(* IEC 61131-3 sources: PLC61131Repos/BZ172Lab/HMIRemote (part 2) *)

	UNTIL pagID <> 16#00
	END_REPEAT;

END_FUNCTION_BLOCK

FUNCTION_BLOCK RefrUnit

	VAR_EXTERNAL
	guiCallStack : ARRAY[ 0..9 ] OF UINT;
	giStackPtr : INT;
	fbUnitString_10 : Static01;
	fbUnitEdit_9 : EditBox01;
	fbUnitEdit_12 : EditBox01;
	fbUnitEdit_13 : EditBox01;
	fbUnitEdit_14 : EditBox01;
	fbUnitEdit_15 : EditBox01;
	fbRefrEvaporatorFan : RefrEvaporatorFan;
	$waitRefresh : BOOL;
	END_VAR

	VAR
	res : USINT;
	pagID : UINT;
	n : USINT;
	iSP : INT;
	pDC : UDINT;
	rx1 : UINT;
	ry1 : UINT;
	rx2 : UINT;
	ry2 : UINT;
	END_VAR

	{CODE:ST}

	REPEAT

		(* Locking the video *)
		res := Video_Lock( res );

		(* Testing if page has changed *)
		pagID := guiCallStack[ giStackPtr ];

		IF pagID = 16#04 THEN

			(* the refresh task is arrived *)
			$waitRefresh := FALSE;

			(* *** REFRESH PAGE CONTROLS *** *)
			IF fbUnitEdit_9.accMode <> kACS_MODIFY THEN
				fbUnitEdit_9();
			END_IF;
			fbUnitEdit_12();
			fbUnitEdit_13();
			fbUnitEdit_14();
			fbUnitEdit_15();

			(* *** REFRESHING BACKGROUND ITEMS *** *)
			(* Cursor across the call stack *)
			iSP := giStackPtr;

			(* *** REFRESHING PARENT BACKGROUND ITEMS *** *)

		END_IF;

		(* Unlocking the video *)
		res := Video_Unlock( res );

		(* Suspending the task *)
		res := Video_Sleep( 50 );

		(* *** MANAGING CHILD WINDOWS AND ALARM MESSAGES *** *)
		IF pagID <> 16#04 THEN
			CASE pagID OF
				16#02:
					fbRefrEvaporatorFan();

			END_CASE;

			(* Re-testing if this page is active *)
			res := Video_Lock( res );
			pagID := guiCallStack[ giStackPtr ];
			res := Video_Unlock( res );
		END_IF;

	UNTIL pagID <> 16#04
	END_REPEAT;

END_FUNCTION_BLOCK

FUNCTION_BLOCK RefrEvaporatorFan

	VAR_EXTERNAL
	guiCallStack : ARRAY[ 0..9 ] OF UINT;
	giStackPtr : INT;
	fbEvaporatorFanString_10 : Static01;
	fbEvaporatorFanString_11 : Static01;
	fbEvaporatorFanString_12 : Static01;
	fbEvaporatorFanString_13 : Static01;
	fbEvaporatorFanEdit_1 : EditBox01;
	fbEvaporatorFanEdit_2 : EditBox01;
	fbEvaporatorFanEdit_3 : EditBox01;
	fbEvaporatorFanEdit_5 : EditBox01;
	fbEvaporatorFanEdit_6 : EditBox01;
	fbEvaporatorFanEdit_7 : EditBox01;
	fbEvaporatorFanEdit_8 : EditBox01;
	fbEvaporatorFanEdit_9 : EditBox01;
	fbRefrCompressor : RefrCompressor;
	$waitRefresh : BOOL;
	END_VAR

	VAR
	res : USINT;
	pagID : UINT;
	n : USINT;
	iSP : INT;
	pDC : UDINT;
	rx1 : UINT;
	ry1 : UINT;
	rx2 : UINT;
	ry2 : UINT;
	END_VAR

	{CODE:ST}

	REPEAT

		(* Locking the video *)
		res := Video_Lock( res );

		(* Testing if page has changed *)
		pagID := guiCallStack[ giStackPtr ];

		IF pagID = 16#02 THEN

			(* the refresh task is arrived *)
			$waitRefresh := FALSE;

			(* *** REFRESH PAGE CONTROLS *** *)
			IF fbEvaporatorFanEdit_1.accMode <> kACS_MODIFY THEN
				fbEvaporatorFanEdit_1();
			END_IF;
			IF fbEvaporatorFanEdit_2.accMode <> kACS_MODIFY THEN
				fbEvaporatorFanEdit_2();
			END_IF;
			IF fbEvaporatorFanEdit_3.accMode <> kACS_MODIFY THEN
				fbEvaporatorFanEdit_3();
			END_IF;
			IF fbEvaporatorFanEdit_5.accMode <> kACS_MODIFY THEN
				fbEvaporatorFanEdit_5();
			END_IF;
			fbEvaporatorFanEdit_6();
			fbEvaporatorFanEdit_7();
			fbEvaporatorFanEdit_8();
			fbEvaporatorFanEdit_9();

			(* *** REFRESHING BACKGROUND ITEMS *** *)
			(* Cursor across the call stack *)
			iSP := giStackPtr;

			(* *** REFRESHING PARENT BACKGROUND ITEMS *** *)

		END_IF;

		(* Unlocking the video *)
		res := Video_Unlock( res );

		(* Suspending the task *)
		res := Video_Sleep( 50 );

		(* *** MANAGING CHILD WINDOWS AND ALARM MESSAGES *** *)
		IF pagID <> 16#02 THEN
			CASE pagID OF
				16#01:
					fbRefrCompressor();

			END_CASE;

			(* Re-testing if this page is active *)
			res := Video_Lock( res );
			pagID := guiCallStack[ giStackPtr ];
			res := Video_Unlock( res );
		END_IF;

	UNTIL pagID <> 16#02
	END_REPEAT;

END_FUNCTION_BLOCK

FUNCTION_BLOCK RefrCompressor

	VAR_EXTERNAL
	guiCallStack : ARRAY[ 0..9 ] OF UINT;
	giStackPtr : INT;
	fbCompressorString_8 : Static01;
	fbCompressorString_9 : Static01;
	fbCompressorString_10 : Static01;
	fbCompressorString_11 : Static01;
	fbCompressorString_12 : Static01;
	fbCompressorEdit_1 : EditBox01;
	fbCompressorEdit_2 : EditBox01;
	fbCompressorEdit_3 : EditBox01;
	fbCompressorEdit_4 : EditBox01;
	fbCompressorEdit_5 : EditBox01;
	fbCompressorEdit_6 : EditBox01;
	fbCompressorEdit_7 : EditBox01;
	fbRefrEXV : RefrEXV;
	$waitRefresh : BOOL;
	END_VAR

	VAR
	res : USINT;
	pagID : UINT;
	n : USINT;
	iSP : INT;
	pDC : UDINT;
	rx1 : UINT;
	ry1 : UINT;
	rx2 : UINT;
	ry2 : UINT;
	END_VAR

	{CODE:ST}

	REPEAT

		(* Locking the video *)
		res := Video_Lock( res );

		(* Testing if page has changed *)
		pagID := guiCallStack[ giStackPtr ];

		IF pagID = 16#01 THEN

			(* the refresh task is arrived *)
			$waitRefresh := FALSE;

			(* *** REFRESH PAGE CONTROLS *** *)
			IF fbCompressorEdit_1.accMode <> kACS_MODIFY THEN
				fbCompressorEdit_1();
			END_IF;
			IF fbCompressorEdit_2.accMode <> kACS_MODIFY THEN
				fbCompressorEdit_2();
			END_IF;
			fbCompressorEdit_3();
			fbCompressorEdit_4();
			fbCompressorEdit_5();
			fbCompressorEdit_6();
			fbCompressorEdit_7();

			(* *** REFRESHING BACKGROUND ITEMS *** *)
			(* Cursor across the call stack *)
			iSP := giStackPtr;

			(* *** REFRESHING PARENT BACKGROUND ITEMS *** *)

		END_IF;

		(* Unlocking the video *)
		res := Video_Unlock( res );

		(* Suspending the task *)
		res := Video_Sleep( 50 );

		(* *** MANAGING CHILD WINDOWS AND ALARM MESSAGES *** *)
		IF pagID <> 16#01 THEN
			CASE pagID OF
				16#06:
					fbRefrEXV();

			END_CASE;

			(* Re-testing if this page is active *)
			res := Video_Lock( res );
			pagID := guiCallStack[ giStackPtr ];
			res := Video_Unlock( res );
		END_IF;

	UNTIL pagID <> 16#01
	END_REPEAT;

END_FUNCTION_BLOCK

FUNCTION_BLOCK RefrEXV

	VAR_EXTERNAL
	guiCallStack : ARRAY[ 0..9 ] OF UINT;
	giStackPtr : INT;
	fbEXVString_10 : Static01;
	fbEXVString_11 : Static01;
	fbEXVString_12 : Static01;
	fbEXVString_13 : Static01;
	fbEXVString_14 : Static01;
	fbEXVEdit_1 : EditBox01;
	fbEXVEdit_2 : EditBox01;
	fbEXVEdit_4 : EditBox01;
	fbEXVEdit_5 : EditBox01;
	fbEXVEdit_6 : EditBox01;
	fbEXVEdit_7 : EditBox01;
	fbEXVEdit_8 : EditBox01;
	fbEXVEdit_9 : EditBox01;
	fbRefrPIDCoefficients : RefrPIDCoefficients;
	$waitRefresh : BOOL;
	END_VAR

	VAR
	res : USINT;
	pagID : UINT;
	n : USINT;
	iSP : INT;
	pDC : UDINT;
	rx1 : UINT;
	ry1 : UINT;
	rx2 : UINT;
	ry2 : UINT;
	END_VAR

	{CODE:ST}

	REPEAT

		(* Locking the video *)
		res := Video_Lock( res );

		(* Testing if page has changed *)
		pagID := guiCallStack[ giStackPtr ];

		IF pagID = 16#06 THEN

			(* the refresh task is arrived *)
			$waitRefresh := FALSE;

			(* *** REFRESH PAGE CONTROLS *** *)
			IF fbEXVEdit_1.accMode <> kACS_MODIFY THEN
				fbEXVEdit_1();
			END_IF;
			IF fbEXVEdit_2.accMode <> kACS_MODIFY THEN
				fbEXVEdit_2();
			END_IF;
			fbEXVEdit_4();
			fbEXVEdit_5();
			fbEXVEdit_6();
			fbEXVEdit_7();
			IF fbEXVEdit_8.accMode <> kACS_MODIFY THEN
				fbEXVEdit_8();
			END_IF;
			fbEXVEdit_9();

			(* *** REFRESHING BACKGROUND ITEMS *** *)
			(* Cursor across the call stack *)
			iSP := giStackPtr;

			(* *** REFRESHING PARENT BACKGROUND ITEMS *** *)

		END_IF;

		(* Unlocking the video *)
		res := Video_Unlock( res );

		(* Suspending the task *)
		res := Video_Sleep( 50 );

		(* *** MANAGING CHILD WINDOWS AND ALARM MESSAGES *** *)
		IF pagID <> 16#06 THEN
			CASE pagID OF
				16#05:
					fbRefrPIDCoefficients();

			END_CASE;

			(* Re-testing if this page is active *)
			res := Video_Lock( res );
			pagID := guiCallStack[ giStackPtr ];
			res := Video_Unlock( res );
		END_IF;

	UNTIL pagID <> 16#06
	END_REPEAT;

END_FUNCTION_BLOCK

FUNCTION_BLOCK RefrPIDCoefficients

	VAR_EXTERNAL
	guiCallStack : ARRAY[ 0..9 ] OF UINT;
	giStackPtr : INT;
	fbPIDCoefficientsString_10 : Static01;
	fbPIDCoefficientsString_11 : Static01;
	fbPIDCoefficientsString_12 : Static01;
	fbPIDCoefficientsEdit_1 : EditBox01;
	fbPIDCoefficientsEdit_2 : EditBox01;
	fbPIDCoefficientsEdit_3 : EditBox01;
	fbPIDCoefficientsEdit_4 : EditBox01;
	fbPIDCoefficientsEdit_5 : EditBox01;
	fbPIDCoefficientsEdit_6 : EditBox01;
	fbPIDCoefficientsEdit_7 : EditBox01;
	fbPIDCoefficientsEdit_8 : EditBox01;
	fbPIDCoefficientsEdit_9 : EditBox01;
	fbRefrPulseAcquisition : RefrPulseAcquisition;
	$waitRefresh : BOOL;
	END_VAR

	VAR
	res : USINT;
	pagID : UINT;
	n : USINT;
	iSP : INT;
	pDC : UDINT;
	rx1 : UINT;
	ry1 : UINT;
	rx2 : UINT;
	ry2 : UINT;
	END_VAR

	{CODE:ST}

	REPEAT

		(* Locking the video *)
		res := Video_Lock( res );

		(* Testing if page has changed *)
		pagID := guiCallStack[ giStackPtr ];

		IF pagID = 16#05 THEN

			(* the refresh task is arrived *)
			$waitRefresh := FALSE;

			(* *** REFRESH PAGE CONTROLS *** *)
			IF fbPIDCoefficientsEdit_1.accMode <> kACS_MODIFY THEN
				fbPIDCoefficientsEdit_1();
			END_IF;
			IF fbPIDCoefficientsEdit_2.accMode <> kACS_MODIFY THEN
				fbPIDCoefficientsEdit_2();
			END_IF;
			IF fbPIDCoefficientsEdit_3.accMode <> kACS_MODIFY THEN
				fbPIDCoefficientsEdit_3();
			END_IF;
			IF fbPIDCoefficientsEdit_4.accMode <> kACS_MODIFY THEN
				fbPIDCoefficientsEdit_4();
			END_IF;
			IF fbPIDCoefficientsEdit_5.accMode <> kACS_MODIFY THEN
				fbPIDCoefficientsEdit_5();
			END_IF;
			IF fbPIDCoefficientsEdit_6.accMode <> kACS_MODIFY THEN
				fbPIDCoefficientsEdit_6();
			END_IF;
			IF fbPIDCoefficientsEdit_7.accMode <> kACS_MODIFY THEN
				fbPIDCoefficientsEdit_7();
			END_IF;
			IF fbPIDCoefficientsEdit_8.accMode <> kACS_MODIFY THEN
				fbPIDCoefficientsEdit_8();
			END_IF;
			IF fbPIDCoefficientsEdit_9.accMode <> kACS_MODIFY THEN
				fbPIDCoefficientsEdit_9();
			END_IF;

			(* *** REFRESHING BACKGROUND ITEMS *** *)
			(* Cursor across the call stack *)
			iSP := giStackPtr;

			(* *** REFRESHING PARENT BACKGROUND ITEMS *** *)

		END_IF;

		(* Unlocking the video *)
		res := Video_Unlock( res );

		(* Suspending the task *)
		res := Video_Sleep( 50 );

		(* *** MANAGING CHILD WINDOWS AND ALARM MESSAGES *** *)
		IF pagID <> 16#05 THEN
			CASE pagID OF
				16#07:
					fbRefrPulseAcquisition();

			END_CASE;

			(* Re-testing if this page is active *)
			res := Video_Lock( res );
			pagID := guiCallStack[ giStackPtr ];
			res := Video_Unlock( res );
		END_IF;

	UNTIL pagID <> 16#05
	END_REPEAT;

END_FUNCTION_BLOCK

FUNCTION_BLOCK RefrPulseAcquisition

	VAR_EXTERNAL
	guiCallStack : ARRAY[ 0..9 ] OF UINT;
	giStackPtr : INT;
	fbPulseAcquisitionString_9 : Static01;
	fbPulseAcquisitionEdit_1 : EditBox01;
	fbPulseAcquisitionEdit_2 : EditBox01;
	fbPulseAcquisitionEdit_3 : EditBox01;
	fbPulseAcquisitionEdit_4 : EditBox01;
	fbPulseAcquisitionEdit_5 : EditBox01;
	fbPulseAcquisitionEdit_6 : EditBox01;
	fbPulseAcquisitionEdit_7 : EditBox01;
	fbPulseAcquisitionEdit_8 : EditBox01;
	$waitRefresh : BOOL;
	END_VAR

	VAR
	res : USINT;
	pagID : UINT;
	n : USINT;
	iSP : INT;
	pDC : UDINT;
	rx1 : UINT;
	ry1 : UINT;
	rx2 : UINT;
	ry2 : UINT;
	END_VAR

	{CODE:ST}

	REPEAT

		(* Locking the video *)
		res := Video_Lock( res );

		(* Testing if page has changed *)
		pagID := guiCallStack[ giStackPtr ];

		IF pagID = 16#07 THEN

			(* the refresh task is arrived *)
			$waitRefresh := FALSE;

			(* *** REFRESH PAGE CONTROLS *** *)
			fbPulseAcquisitionEdit_1();
			fbPulseAcquisitionEdit_2();
			fbPulseAcquisitionEdit_3();
			fbPulseAcquisitionEdit_4();
			fbPulseAcquisitionEdit_5();
			fbPulseAcquisitionEdit_6();
			fbPulseAcquisitionEdit_7();
			fbPulseAcquisitionEdit_8();

			(* *** REFRESHING BACKGROUND ITEMS *** *)
			(* Cursor across the call stack *)
			iSP := giStackPtr;

			(* *** REFRESHING PARENT BACKGROUND ITEMS *** *)

		END_IF;

		(* Unlocking the video *)
		res := Video_Unlock( res );

		(* Suspending the task *)
		res := Video_Sleep( 50 );

	UNTIL pagID <> 16#07
	END_REPEAT;

END_FUNCTION_BLOCK

	(***************************)
	(*                         *)
	(* PARAMETER  FUN. BLOCKS  *)
	(*                         *)
	(***************************)
